{attribute 'qualified_only'}
{attribute 'strict'}
TYPE SerialParity :
(
	None := 0,
	Odd,
	Even,
	Mark,
	Space
);
END_TYPE

(* stored: Version 1.1.0.1, ProductVersion 3.1.4024.3
   DUT SerialParity: Id {1fe467c0-9caa-421e-994b-d32e57a105f4} *)
